TYPE E_CffExitIntent : (
    CFF_EXIT_NONE := 0,
    CFF_EXIT_NORMAL_RETURN := 10,
    CFF_EXIT_NOK_RETURN := 20,
    CFF_EXIT_ABORT_NO_RETURN := 30,
    CFF_EXIT_FAULT_NO_RETURN := 40
); END_TYPE

(* stored: Version 1.1.0.1
   DUT E_CffExitIntent: Id {7FBFD290-60B5-4FCE-8D00-D46650117E64} *)
